FUNCTION_BLOCK TcoLogger EXTENDS TcoObject
VAR
	_buffer : ARRAY[0..1000] OF TcoMessage;
	_plcCarret : INT;
	_minLoggingLevel : eMessageCategory := eMessageCategory.Notification;
END_VAR

VAR CONSTANT
	MESSAGE_BUFFER_LENGHT : INT := 1000;
END_VAR

METHOD Push
VAR_INPUT
	inMessage : TcoMessage;
END_VAR
IF(inMessage.Category < THIS^._minLoggingLevel) THEN
	RETURN;
END_IF

IF(_plcCarret > MESSAGE_BUFFER_LENGHT) THEN
	_plcCarret := 0;
END_IF

_buffer[_plcCarret] := inMessage;
_buffer[_plcCarret].ExpectDequeing := TRUE;
_buffer[_plcCarret].Cycle := THIS^.Context.StartCycleCount;

_plcCarret := _plcCarret + 1;
END_METHOD

END_FUNCTION_BLOCK

(* stored: Version 1.1.0.1, ProductVersion 3.1.4024.9
   POU TcoLogger: Id {e93d64b3-7935-00d0-1165-0e260b788c79}, SpecialFunc None
   Method Push: Id {fc2f2ea9-87af-0452-32db-ced92ed04c01} *)
